# EPICS substitutions: iocBoot/ioc13Keithley_DACpiezo/Instek.substitutions
file "$(IP)/ipApp/Db/Instek.db" { pattern
{P,          R,       PORT,    LOPR,  HOPR,   PREC,   SCAN,        CONFIG_SCAN}
{13DAC_piezo:, Instek1,  serial2,    0,  2000,   1,     ".5 second", "5 second"}
{13DAC_piezo:, Instek1,  serial3,    0,  2000,   1,     ".5 second", "5 second"}
{13DAC_piezo:, Instek1,  serial4,    0,  2000,   1,     ".5 second", "5 second"}
}
